// TIA Portal V18 export
DATA_BLOCK "SS1_754A1_16DI_DI_Vars"   // DB11061
{ S7_Optimized_Access := 'FALSE' }
VERSION : 0.1
// stored: AutoNumber false, DBAccessibleFromOPCUA true, IsOnlyStoredInLoadMemory false, IsWriteProtectedInAS false
   VAR
      DI1 : "UDT_DIadv";   // AHU NF Термостат загр. замерз. (2.50)
      DI2 : "UDT_DIadv";   // AHU NF Авто. режим пр. вент. (2.200)
      DI3 : "UDT_DIadv";   // AHU NF 1-шв. пр. вент. (2.200)
      DI4 : "UDT_DIadv";   // AHU NF 2-шв. пр. вент. (2.200)
      DI5 : "UDT_DIadv";   // AHU NF Тепл. реле. 1-шв. пр. вент. (2.200)
      DI6 : "UDT_DIadv";   // AHU NF Тепл. реле. 2-шв. пр. вент. (2.200)
      DI7 : "UDT_DIadv";   // AHU NF Несправність пр. вент. (2.200)
      DI8 : "UDT_DIadv";   // AHU NF Інд. сервісний вимикач. пр. вент. (2.200)
      DI9 { S7_SetPoint := 'True'} : "UDT_DIadv";   // AHU NF Несправність клиновий ркмінь пр. вент. (2.54)
      DI10 { S7_SetPoint := 'True'} : "UDT_DIadv";   // AHU NF Забруднення пр. фільтру (2.53)
      DI11 { S7_SetPoint := 'True'} : "UDT_DIadv";   // AHU NF Робота цирк. насос (2.201)
      DI12 { S7_SetPoint := 'True'} : "UDT_DIadv";   // AHU NF Авто режим цирк. насос (2.201)
      DI13 { S7_SetPoint := 'True'} : "UDT_DIadv";   // AHU NF Несправність цирк. насос (2.201)
      DI14 { S7_SetPoint := 'True'} : "UDT_DIadv";   // HS Робота вн. насос К1 (10.209)
      DI15 { S7_SetPoint := 'True'} : "UDT_DIadv";   // HS Перегрів вн. насос К1 (10.209) термоконтакт
      DI16 { S7_SetPoint := 'True'} : "UDT_DIadv";   // HS Робота вн. насос К2 (10.210)
   END_VAR
BEGIN
   DI1.cFuncSystemID := 100;
   DI1.cFuncVar := 1;
   DI2.cFuncSystemID := 100;
   DI2.cFuncVar := 3;
   DI5.cFuncSystemID := 100;
   DI5.cFuncVar := 5;
   DI6.cFuncSystemID := 100;
   DI6.cFuncVar := 6;
END_DATA_BLOCK
